Omron Sysmac Studio project OEEF_FS_lib_1_2_2 (Sysmac Studio 1.44.0.64015, LibraryProject)

# Controller new_Controller_0: NX1P2-1040DT1 version 1.21
Task PrimaryTask (priority 4, period or condition 2000): Programme0

TYPE nsAxisControl\eMoveMode : (Relative := 0, Absolute := 1); END_TYPE
TYPE nsAxisControl\eCurveType : (Poly5 := 0, Poly3 := 1, Straight := 2, NoCurve := 9999); END_TYPE
TYPE nsAxisControl\eTypeOfCmd : (CancelMC_Sync := -5, CancelCam := -3, CancelTrack := -2, NoCde := 9999, PolyMvt := 1, Track := 2, Cam := 3, WarmStart := 4, MC_Sync := 5); END_TYPE
TYPE nsAxisControl\stAxisControl : STRUCT
    MasterPosition : nsAxisControl\stMasterPosition;
    MasterAxis : _sAXIS_REF;
    Move : nsAxisControl\stMove;
    Track : nsAxisControl\stTrack;
    Cam : nsAxisControl\stCam;
    Kinematic : nsAxisControl\stKinematic;
    Flags : nsAxisControl\stFlags;
    Monitoring : nsAxisControl\stMonitoring;
    MC_MoveJog : nsAxisControl\stMC_MoveJog;
    MC_SetPosition : nsAxisControl\stMC_SetPosition;
    MC_Power : nsAxisControl\stMC_Power;
    MC_Home : nsAxisControl\stMC_Home;
END_STRUCT END_TYPE
TYPE nsAxisControl\stMC_Power : STRUCT
    Enable : BOOL;
    Status : BOOL;
    Busy : BOOL;
    Error : BOOL;
    ErrorID : WORD;
END_STRUCT END_TYPE
TYPE nsAxisControl\stMC_MoveJog : STRUCT
    PositiveEnable : BOOL;
    NegativeEnable : BOOL;
    Velocity : LREAL;
    Acceleration : LREAL;
    Deceleration : LREAL;
    Busy : BOOL;
    CommandAborted : BOOL;
    Error : BOOL;
    ErrorID : WORD;
END_STRUCT END_TYPE
TYPE nsAxisControl\stMC_SetPosition : STRUCT
    Execute : BOOL;
    Position : LREAL;
    ReferenceType : _eMC_REFERENCE_TYPE;
    Relative : BOOL;
    ExecutionMode : _eMC_EXECUTION_MODE;
    Done : BOOL;
    Busy : BOOL;
    CommandAborted : BOOL;
    Error : BOOL;
    ErrorID : WORD;
END_STRUCT END_TYPE
TYPE nsAxisControl\stMC_Home : STRUCT
    Execute : BOOL;
    Done : BOOL;
    Busy : BOOL;
    CommandAborted : BOOL;
    Error : BOOL;
    ErrorID : WORD;
END_STRUCT END_TYPE
TYPE nsAxisControl\stMasterPosition : STRUCT
    NotFrom_sAXIS_REF : BOOL;
    ExternalVariable : LREAL;
END_STRUCT END_TYPE
TYPE nsAxisControl\stMove : STRUCT
    Pos : LREAL;
    Dist : LREAL;
    Tim : LREAL;
    Accel : LREAL;
    Decel : LREAL;
    PolyType : nsAxisControl\eCurveType;
    Mode : nsAxisControl\eMoveMode;
    SetT_In : LREAL;
    SetT_Out : LREAL;
    T_InDone : BOOL;
    T_OutDone : BOOL;
    Exe : BOOL;
END_STRUCT END_TYPE
TYPE nsAxisControl\stTrack : STRUCT
    Conveyor_Vel : LREAL;
    Pos : LREAL;
    Tim : LREAL;
    TimStop : LREAL;
    Accel : LREAL;
    Decel : LREAL;
    PolyType : nsAxisControl\eCurveType;
    SetT_In : LREAL;
    T_InDone : BOOL;
    Exe : BOOL;
    Cancel : BOOL;
END_STRUCT END_TYPE
TYPE nsAxisControl\stCam : STRUCT
    Profile : ARRAY[0..10] OF nsAxisControl\stNodes;
    FirstProfile : INT;
    WarmStartMasterPos : LREAL;
    WarmStartSlavePos : LREAL;
    WarmStartSlavePosRequest : BOOL;
    Exe : BOOL;
    Cancel : BOOL;
END_STRUCT END_TYPE
TYPE nsAxisControl\stNodes : STRUCT
    Node : ARRAY[0..10] OF nsAxisControl\stNode;
END_STRUCT END_TYPE
TYPE nsAxisControl\stNode : STRUCT
    MasterAxisPos : LREAL;
    SlaveAxisPos : LREAL;
    CurveTypeBefore : nsAxisControl\eCurveType;
    StartingSlope : LREAL;
    EndingSlope : LREAL;
    PreviousProfile : INT;
    NextProfile : INT;
END_STRUCT END_TYPE
TYPE nsAxisControl\stKinematic : STRUCT
    Start : BOOL;
    Stop : BOOL;
    InvKin_in : LREAL;
    InvKin_out : LREAL;
    DirKin_in : LREAL;
    DirKin_out : LREAL;
END_STRUCT END_TYPE
TYPE nsAxisControl\stFlags : STRUCT
    Done : BOOL;
    Synchronising : BOOL;
    Synchronised : BOOL;
END_STRUCT END_TYPE
TYPE nsAxisControl\stMonitoring : STRUCT
    PositioningCmd : LREAL;
    Axis_Act_Pos_MCS : LREAL;
    TypeOfCmd : nsAxisControl\eTypeOfCmd;
    TypeOfCtrlMode : nsAxisControl\eTypeOfCtrlMode;
END_STRUCT END_TYPE
TYPE nsAxisControl\eTypeOfCtrlMode : (ExtKinOff := 0, ExtKinOn := 1, NoCtrlMode := 9999); END_TYPE

TYPE nsKinematics\sKinInOut : STRUCT
    KinSpec : nsKinematics\stSpec;
    Cartesian : nsKinematics\sCartesian;
    Axis : nsKinematics\sAxis;
    KinSize : nsKinematics\stSize;
END_STRUCT END_TYPE
TYPE nsKinematics\stSpec : STRUCT
    KinType : nsKinematics\eKinType;
    KinDir : nsKinematics\eDirInv;
    SCARA : nsKinematics\stSCARA;
END_STRUCT END_TYPE
TYPE nsKinematics\sCartesian : STRUCT
    Cmd_Component : ARRAY[0..2] OF LREAL;
    Act_Component : ARRAY[0..2] OF LREAL;
END_STRUCT END_TYPE
TYPE nsKinematics\sAxis : STRUCT
    A_Cmd : ARRAY[0..9] OF LREAL;
    A_Act : ARRAY[0..9] OF LREAL;
END_STRUCT END_TYPE
TYPE nsKinematics\eKinType : (H_Bot_XY := 0, SCARA := 1); END_TYPE
TYPE nsKinematics\eDirInv : (Direct := 0, Inverse := 1); END_TYPE
TYPE nsKinematics\stSize : STRUCT
    NbOfCoordinates : INT;
    NbOfAxis : INT;
END_STRUCT END_TYPE
TYPE nsKinematics\stSCARA : STRUCT
    Len1 : LREAL;
    Len2 : LREAL;
END_STRUCT END_TYPE

PROGRAM Programme0

(* Section Section0: ladder, written here as Structured Text *)
END_PROGRAM

FUNCTION fPolyTimesNeeded : BOOL
(* Time needed to achieve a movement depending of the curve type and the acceleration or the speed fixed. To do for instance a speed or an acceleration limit. *)
VAR_INPUT
    CurveType : nsAxisControl\eCurveType;
    Distance : LREAL;
    AccDefined : LREAL;
    SpeedDefined : LREAL;
END_VAR
VAR_OUTPUT
    TNeededToAcc : LREAL;
    TNeededToSpeed : LREAL;
END_VAR
(*
*******************************************
*		  Calcule le temps nécessaire			*
*	 pour effectuer un trajet avec une		*
*	accélération ou une vitesse définie		*
*******************************************
*)

CASE CurveType OF
	
	Poly5 :
	// AccDefined exprimée en unité/sec2
	TNeededToAcc:=SQRT(5.8*Distance/AccDefined);

	// SpeedDefined exprimée en unité/sec
	TNeededToSpeed:=1.9*Distance/SpeedDefined;
	
	Poly3 :
	// AccDefined exprimée en unité/sec2
	TNeededToAcc:=SQRT(6*Distance/AccDefined);

	// SpeedDefined exprimée en unité/sec
	TNeededToSpeed:=1.5*Distance/SpeedDefined;
	
END_CASE;
END_FUNCTION

FUNCTION fKinematics : BOOL
(* Normal and inverse tranforms : / - H-Bot XY / - SCARA *)
VAR
    AC : LREAL;
    BAC : LREAL;
    ABC : LREAL;
    angle : LREAL;
    len1 : LREAL;
    len2 : LREAL;
    j2 : LREAL;
    j1 : LREAL;
    x : LREAL;
    y : LREAL;
    z : LREAL;
END_VAR
VAR_IN_OUT
    KinInOut : nsKinematics\sKinInOut;
END_VAR
(*
*******************************************
*		  			Transformées						*
*	 			directes et inverses					*
*******************************************
*)

CASE KinInOut.KinSpec.KinType OF
	(* H-Bot XY *)
	H_Bot_XY :
	KinInOut.KinSize.NbOfCoordinates:=2;				// XY
	KinInOut.KinSize.NbOfAxis:=2;							// A0 et A1

	IF KinInOut.KinSpec.KinDir=Direct THEN
		// Direct
		KinInOut.Cartesian.Act_Component[0]:=(KinInOut.Axis.A_Act[0]+KinInOut.Axis.A_Act[1])*0.5;							// positions actuelle X
		KinInOut.Cartesian.Act_Component[1]:=(KinInOut.Axis.A_Act[0]-KinInOut.Axis.A_Act[1])*0.5;							// positions actuelle Y
	ELSE
		// Inverse
		KinInOut.Axis.A_Cmd[0]:=KinInOut.Cartesian.Cmd_Component[0]+KinInOut.Cartesian.Cmd_Component[1];	// Position de commande axe A0
		KinInOut.Axis.A_Cmd[1]:=KinInOut.Cartesian.Cmd_Component[0]-KinInOut.Cartesian.Cmd_Component[1];	// Position de commande axe A1
	END_IF;	

	(* SCARA *)
	SCARA :
	KinInOut.KinSize.NbOfCoordinates:=3;				// XYZ
	KinInOut.KinSize.NbOfAxis:=3;							// A0 à A2
	
	len1:=KinInOut.KinSpec.SCARA.Len1;					// Longueur du bras
	len2:=KinInOut.KinSpec.SCARA.Len2;					// Longueur de l'avant bras	
	
	IF KinInOut.KinSpec.KinDir=Direct THEN
		// Direct
		j1:=KinInOut.Axis.A_Act[0];								// Angle actuel de l'épaule
		j2:=KinInOut.Axis.A_Act[1];								// Angle actuel du coude
		
		AC:=SQRT(len1*len1+len2*len2-2*len1*len2*COS(DegToRad(j2)));
		BAC:=RadToDeg(ACOS((len1*len1+AC*AC-len2*len2)/(2*len1*AC)));	
		angle:=j1-BAC;
		
		fBaseCoords(AC, angle, KinInOut.Cartesian.Act_Component[0], KinInOut.Cartesian.Act_Component[1]);			// positions actuelles X et Y 
		KinInOut.Cartesian.Act_Component[2]:=KinInOut.Axis.A_Act[2];																		// position actuelle Z 
		
	ELSE
		// Inverse
		x:=KinInOut.Cartesian.Cmd_Component[0];	// Position de commande X
		y:=KinInOut.Cartesian.Cmd_Component[1];	// Position de commande Y
		z:=KinInOut.Cartesian.Cmd_Component[2];	// Position de commande Z
		
		AC:=SQRT(x*x+y*y);
		ABC:=RadToDeg(ACOS((len1*len1+len2*len2-AC*AC)/(2*len1*len2)));
		
		KinInOut.Axis.A_Cmd[0]:=ABC;						// Angle de commande axe 0 (épaule)
		
		IF x>0 AND y>0 THEN										// Angle de commande axe 1 (coude)
			KinInOut.Axis.A_Cmd[1]:=RadToDeg(ACOS(AC/x));
		ELSIF x>0 AND y<0 THEN
			KinInOut.Axis.A_Cmd[1]:=180-RadToDeg(ACOS(AC/x));
		ELSIF x<0 AND y<0 THEN
			KinInOut.Axis.A_Cmd[1]:=180+RadToDeg(ACOS(AC/x));
		ELSE
			KinInOut.Axis.A_Cmd[1]:=360-RadToDeg(ACOS(AC/x));
		END_IF;
		
		KinInOut.Axis.A_Cmd[2]:=z;								// Position de commande axe 2 (vertical)
	END_IF;
END_CASE;
	
END_FUNCTION

FUNCTION fTicksQCalc : LINT
(* Calculation of the quantity of ticks depending of the time of the movement *)
VAR
    TaskPeriod_msec : LINT;
END_VAR
VAR_INPUT
    Tmvt : LREAL;
END_VAR
(*
*******************************************
*		  			Calcul le nombre					*
*	 				de tops d'horloge				*
*******************************************
*)

// Suivant le temps de cycle de la tâche principale
TaskPeriod_msec:= TimeToNanoSec(GetMyTaskInterval())/1000000;

// Suivant le temps du mouvement en secondes
fTicksQCalc:=LREAL_TO_LINT(Tmvt)*1000/TaskPeriod_msec;
END_FUNCTION

FUNCTION fPoly5 : LREAL
(* Polynomial of the 5th order *)
VAR
    a : LREAL;
    b : LREAL;
    c : LREAL;
    d : LREAL;
    e : LREAL;
    f : LREAL;
    K : LREAL;
    xSq : LREAL;
END_VAR
VAR_INPUT
    v0 : LREAL;  (* Vitesse initiale *)
    v1 : LREAL;  (* Vitesse finale *)
    a0 : LREAL;
    a1 : LREAL;
    x : LREAL;
    Offset : LREAL;
    TargetDist : LREAL;
END_VAR
(*
*******************************************
*		  				Polynôme 5						*
*******************************************
*)

// Coéficients 
a:=6.0-3.0*(v0+v1)+((a1-a0)/2.0);
b:=-15.0+8.0*v0+7.0*v1+(3.0*a0/2.0)-a1;
c:=10.0-6.0*v0-4.0*v1-(3.0*a0/2.0)+(a1/2.0);
d:=a0/2.0;
e:=v0;
f:=Offset;
K:=TargetDist;

// Carré de x
xSq:=x*x;

// Position=ax5+bx4+cx3+dx2+ex+f
fPoly5:=f+(K*(a*(xSq*xSq*x)+b*(xSq*xSq)+c*(xSq*x)+d*(xSq)+e*x));
END_FUNCTION

FUNCTION fPoly3 : LREAL
(* Polynomial of the 3th order *)
VAR
    a : LREAL;
    b : LREAL;
    c : LREAL;
    d : LREAL;
    K : LREAL;
    xSq : LREAL;
END_VAR
VAR_INPUT
    v0 : LREAL;  (* Vitesse initiale *)
    v1 : LREAL;  (* Vitesse finale *)
    x : LREAL;
    Offset : LREAL;
    TargetDist : LREAL;
END_VAR
(*
*******************************************
*		  				Polynôme 3						*
*******************************************
*)

// Coéficients 
a:=-2.0+v0+v1;
b:=3.0-2.0*v0-v1;
c:=v0;
d:=Offset;
K:=TargetDist;
		
// Carré de x
xSq:=x*x;

// Position=ax3+bx2+cx+d
fPoly3:=d+(K*(a*(xSq*x)+b*(xSq)+c*x));
END_FUNCTION

FUNCTION fPoly2 : LREAL
(* Polynomial of the 2th order *)
VAR
    a : LREAL;
    b : LREAL;
    c : LREAL;
    xSq : LREAL;
END_VAR
VAR_INPUT
    v0 : LREAL;  (* Vitesse initiale *)
    v1 : LREAL;  (* Vitesse finale *)
    x : LREAL;
    Offset : LREAL;
    TargetDist : LREAL;
END_VAR
(*
*******************************************
*		  				Polynôme 2						*
*******************************************
*)

// Coéfficients
a:=v1-v0;
b:=v0;
c:=Offset;

// Carré de x
xSq:=x*x;

// Position=0,5*ax2+bx+c (primitive d'une droite ax+b)
fPoly2:=(TargetDist*((0.5*a*(xSq)+b*x)))+c;
END_FUNCTION

FUNCTION fStraight : LREAL
(* Straight *)
VAR
    a : LREAL;
    b : LREAL;
END_VAR
VAR_INPUT
    x : LREAL;
    Offset : LREAL;
    TargetDist : LREAL;
END_VAR
(*
*******************************************
*		  					Droite							*
*******************************************
*)

// Coéficients 
a:=TargetDist;
b:=Offset;

// Position=ax+b
fStraight:=a*x+b;
END_FUNCTION

FUNCTION fBaseCoords : BOOL
(* Return coordinates of second joint *)
VAR_INPUT
    length : LREAL;
    angle : LREAL;
END_VAR
VAR_OUTPUT
    x : LREAL;
    y : LREAL;
END_VAR
(*
*******************************************
*		Calcule les coordonnées	XY			*
*		du deuxième joint articulaire			*
*******************************************
*)

IF angle<=90 THEN
	// Premier quadrant
	x:=length*COS(DegToRad(angle));
	y:=length*SIN(DegToRad(angle));
ELSIF angle>90 AND angle<=180 THEN
	// Deuxième quadrant
	x:=-length*COS(DegToRad(180-angle));
	y:=length*SIN(DegToRad(180-angle));
ELSIF angle>180 AND angle<=270 THEN
	// Troisième quadrant
	x:=-length*COS(DegToRad(180-angle));
	y:=-length*SIN(DegToRad(180-angle));
ELSE
	// Quatrième quadrant
	x:=length*COS(DegToRad(360-angle));
	y:=-length*SIN(DegToRad(360-angle));
END_IF;
END_FUNCTION

FUNCTION_BLOCK AxisControl
(* - Cam (multi profiles and Warm start) / - Move abs or rel (pos + time) by polynomials curves (3 & 5) / - Tracking a conveyor / - Blending two axis (T_In & T_Out) / 2. Polynomial 2 for a linear deceleration of the speed in case of track cancelling / 3. Some PLCopen functions nested / 4. Exernal kinematics binding *)
VAR
    FBi_SyncMov : MC_SyncMoveAbsolute;
    FBi_SyncStop : MC_Stop;
    FBe_SetPosition : MC_SetPosition;
    FBe_Home : MC_Home;
    FBi_ReadAxisMasterParam : MC_ReadAxisParameter;
    FBi_ReadAxisSlaveParam : MC_ReadAxisParameter;
    FBe_Power : MC_Power;
    Edge1 : R_TRIG;
    Edge2 : R_TRIG;
    Edge3 : R_TRIG;
    Edge4 : R_TRIG;
    Edge5 : R_TRIG;
    Edge6 : R_TRIG;
    Edge7 : R_TRIG;
    Edge8 : R_TRIG;
    Edge9 : R_TRIG;
    Edge10 : R_TRIG;
    Edge11 : R_TRIG;
    Edge12 : R_TRIG;
    TypeOfCmd : nsAxisControl\eTypeOfCmd;
    TargetDist : LREAL;
    TargetSpeed : LREAL;
    UpExecMvt : BOOL;
    UpExecTrack : BOOL;
    UpExecCam : BOOL;
    UpCancelTrack : BOOL;
    Phase : INT;
    Tick : LINT;
    TicksQ : LINT;
    Offset : LREAL;
    x : LREAL;
    v0 : LREAL;  (* Vitesse initiale *)
    v1 : LREAL;  (* Vitesse finale *)
    LastSpeed : LREAL;
    DistStop : LREAL;
    SyncErr : BOOL;
    SyncErrID : WORD;
    SyncStopErrID : WORD;
    UpKinOn : BOOL;
    UpKinOff : BOOL;
    UpCancelCam : BOOL;
    MasterDistDone : LREAL;
    a1 : LREAL;
    a0 : LREAL;
    FBe_MovJog : MC_MoveJog;
    LastPosSlave : LREAL;
    LastPosMaster : LREAL;
    ReadAxisMasterPParam : _sAXIS_PARAM;
    ReadAxisMasterParameterErr : BOOL;
    ReadAxisMasterParameterErrID : WORD;
    ReadAxisSlavePParam : _sAXIS_PARAM;
    ReadAxisSlaveParameterErr : BOOL;
    ReadAxisSlaveParameterErrID : WORD;
    CamSettingError : BOOL;
    NodesNbMax : INT;
    CurrentSeg : INT;
    Loop : INT;
    X0 : LREAL;
    X1 : LREAL;
    Y0 : LREAL;
    Y1 : LREAL;
    SegmentPolyType : nsAxisControl\eCurveType;
    MasterDist : LREAL;
    SegmentsNb : INT;
    SyncStopErr : BOOL;
    NodesNb : INT;
    UpWarmStartPosReq : BOOL;
    WarmStartCalculation : BOOL;
    v1CamSetting : LREAL;
    v0CamSetting : LREAL;
    Edge10_Q : BOOL;
    Edge10_Clk : BOOL;
    a0CamSetting : LREAL;
    a1CamSetting : LREAL;
    ScannedSeg : INT;
    SetPositionErr : BOOL;
    SetPositionErrID : WORD;
    FBi_SetPosition : MC_SetPosition;
    ProfileToApply : INT := 0;
    ProfilesNb : INT;
    ProfilesNbMax : INT;
    UpCamBeginning : BOOL;
    CamSettingErrorType : STRING[50];
    KinIn : LREAL;
    KinOut : LREAL;
    TypeOfCtrlMode : nsAxisControl\eTypeOfCtrlMode;
    Gen : LREAL;
    Conveyor_Pos : LREAL;
    TaskPeriod_msec_LREAL : LREAL;
    MasterPosition : LREAL;
END_VAR
VAR_INPUT
    Dummy : BOOL;
END_VAR
VAR_OUTPUT
    Error : BOOL;
END_VAR
VAR_IN_OUT CONSTANT
    Axis : _sAXIS_REF;
END_VAR
VAR_IN_OUT
    IO : nsAxisControl\stAxisControl;
END_VAR
VAR_OUTPUT
    ErrorMsg : STRING[80];
END_VAR
(*
*******************************************
*					OEEF - F.SIMON					*
*******************************************
*)

Edge1(IO.Move.Exe,UpExecMvt);															// Commande de mouvement polynômial
Edge2(IO.Track.Exe,UpExecTrack);														// Commande de tracking
Edge3(IO.Track.Cancel,UpCancelTrack);												// Commande d'annulation de tracking
Edge4(IO.Cam.Exe,UpExecCam);															// Commande de mise en came
Edge5(IO.Cam.Cancel,UpCancelCam);													// Commande d'annulation de came
Edge6(IO.Cam.WarmStartSlavePosRequest,UpWarmStartPosReq);		// Commande de Warmstart
Edge7(IO.Kinematic.Start,UpKinOn);													// Commande d'activation de la kinematic
Edge8(IO.Kinematic.Stop,UpKinOff);													// Commande de désactivation de la kinematic


(*
*******************************************
*					Type d'axe maître				*
*******************************************
*)
IF IO.MasterPosition.NotFrom_sAXIS_REF THEN
	MasterPosition:=IO.MasterPosition.ExternalVariable;
ELSE
	MasterPosition:=IO.MasterAxis.Act.Pos;
END_IF;


(*
*******************************************
*		Commande de tracking active		*
*******************************************
*)
IF TypeOfCmd=Track THEN
	// Calcul l'avance du convoyeur
	TaskPeriod_msec_LREAL:= LINT_TO_LREAL(TimeToNanoSec(GetMyTaskInterval())/1000000);
	Conveyor_Pos:=Conveyor_Pos+IO.Track.Conveyor_Vel*(TaskPeriod_msec_LREAL/1000);
	// Polynôme en cours : lecture de la position et de la vitesse du maître pour le raccordement en fin de polynôme
	LastPosMaster:=Conveyor_Pos;					// Position du maître à l'instant
	TargetSpeed:=IO.Track.Conveyor_Vel;			// Vitesse du maître à l'instant
	TargetDist:=LastPosMaster-LastPosSlave; 	// Distance à parcourir depuis l'origine du tracking
	IF IO.Flags.Synchronised THEN
	// Polynôme terminé : synchronisation maître/esclave (following)
		FBi_SyncMov.Position:=Conveyor_Pos;
	END_IF;
END_IF;


(*
*******************************************
*			Commande 	de came					*
*			ou de warmstart active 				*
*******************************************
*)
IF TypeOfCmd=Cam OR TypeOfCmd=WarmStart THEN
	// Profil à appliquer
	Edge9(TRUNC(MasterPosition)=IO.Cam.Profile[ProfileToApply].Node[0].MasterAxisPos,UpCamBeginning);
	IF UpCamBeginning THEN
		IF CurrentSeg=0 THEN
			ProfileToApply:=IO.Cam.Profile[ProfileToApply].Node[0].PreviousProfile; 				// Recule
		ELSE
			ProfileToApply:=IO.Cam.Profile[ProfileToApply].Node[NodesNb-1].NextProfile;	// Avance
		END_IF;
	END_IF;
	
	// Dans le cas d'un WarmStart le profil est imposé car il ne peut être déterminé automatiquement
	IF TypeOfCmd=WarmStart THEN
		ProfileToApply:=IO.Cam.FirstProfile;
	END_IF;

	// Comptage du nombre de noeuds du profil appliqué
	NodesNb:=1;
	WHILE IO.Cam.Profile[ProfileToApply].Node[NodesNb].MasterAxisPos<>0
		DO
		NodesNb:=NodesNb+1;
	END_WHILE;
	
	// Comptage du nombre total de profils
	ProfilesNb:=0;
	REPEAT
		ProfilesNb:=ProfilesNb+1;
	UNTIL IO.Cam.Profile[ProfilesNb].Node[1].MasterAxisPos=0
	END_REPEAT;
	
	// Nombre de segments de la came
	SegmentsNb:=NodesNb-1;
		
	// Evolution du segment en cours
	CASE TypeOfCmd OF
		Cam :
		FOR ScannedSeg:=0 TO SegmentsNb-1 DO
			IF MasterPosition>=IO.Cam.Profile[ProfileToApply].Node[ScannedSeg].MasterAxisPos AND MasterPosition<IO.Cam.Profile[ProfileToApply].Node[ScannedSeg+1].MasterAxisPos THEN
				CurrentSeg:=ScannedSeg;
			END_IF;
		END_FOR;
		WarmStart :
		FOR ScannedSeg:=0 TO SegmentsNb-1 DO
			IF IO.Cam.WarmStartMasterPos>=IO.Cam.Profile[ProfileToApply].Node[ScannedSeg].MasterAxisPos AND IO.Cam.WarmStartMasterPos<IO.Cam.Profile[ProfileToApply].Node[ScannedSeg+1].MasterAxisPos THEN
				CurrentSeg:=ScannedSeg;
			END_IF;
		END_FOR;	
	END_CASE;

	// Paramètres du polynôme dans le segment en cours
	X0:=IO.Cam.Profile[ProfileToApply].Node[CurrentSeg].MasterAxisPos;										// Abscisse de début
	Y0:=IO.Cam.Profile[ProfileToApply].Node[CurrentSeg].SlaveAxisPos;											// Ordonnée de début
	X1:=IO.Cam.Profile[ProfileToApply].Node[CurrentSeg+1].MasterAxisPos;									// Abscisse de fin
	Y1:=IO.Cam.Profile[ProfileToApply].Node[CurrentSeg+1].SlaveAxisPos;									// Ordonnée de fin
	MasterDist:=X1-X0;																														// Distance de la composante X
	TargetDist:=Y1-Y0;																														// Distance de la composante Y
	Offset:=Y0;																																	// Offset de départ

 	CASE TypeOfCmd OF
		Cam : MasterDistDone:=MasterPosition-X0;																			// Distance parcourue par le maître
		WarmStart : MasterDistDone:=IO.Cam.WarmStartMasterPos-X0;
 	END_CASE;
 
	SegmentPolyType:=IO.Cam.Profile[ProfileToApply].Node[CurrentSeg+1].CurveTypeBefore;		// Type de profil
	v0CamSetting:=IO.Cam.Profile[ProfileToApply].Node[CurrentSeg+1].StartingSlope;					// Pente de raccordement de la vitesse de début de segment
	v1CamSetting:=IO.Cam.Profile[ProfileToApply].Node[CurrentSeg+1].EndingSlope;					// Pente de raccordement de la vitesse de fin de segment
	//a0CamSetting:=?																														// Pente de raccordement de l'accélération de début de segment
	//a1CamSetting:=?																														// Pente de raccordement de l'accélération de fin de segment

	// Arrêt du calcul de la position théorique de l'esclave pour le WarmStart
	IF WarmStartCalculation THEN
		WarmStartCalculation:=FALSE;
	END_IF;
END_IF;


(*
*******************************************
*				Mode kinematic actif				*
*******************************************
*)
IF TypeOfCtrlMode=ExtKinOn THEN
	// Envoi le calcul du générateur vers la kinematic
	KinIn:=Gen;
	// Désactive le mode External kinematic en cas d'erreur du MC_SyncMoveAbsolute
	IF FBi_SyncMov.Error THEN
		TypeOfCtrlMode:=NoCtrlMode;
	END_IF;

	// Envoi la commande de position MCS à la kinématic inverse
	IO.Kinematic.InvKin_in:=KinIn;
	// Récupère la commande de position ACS
	KinOut:=IO.Kinematic.InvKin_out;

	// Envoi la position actuelle ACS à la kinématic directe
	IO.Kinematic.DirKin_in:=Axis.Act.Pos;
	// Récupère la position actuelle MCS
	IO.Monitoring.Axis_Act_Pos_MCS:=IO.Kinematic.DirKin_out;
END_IF;


(*
*******************************************
*			Mode kinematic inactif				*
*******************************************
*)
IF TypeOfCtrlMode=ExtKinOff THEN
	// Envoi le calcul du générateur vers la kinematic
	KinIn:=Gen;
	// ACS=MCS
	KinOut:=KinIn;
	IO.Monitoring.Axis_Act_Pos_MCS:=Axis.Act.Pos;
END_IF;


(*
*******************************************
*						Générateur						*
*******************************************
*)
CASE Phase OF
	
	0 : // COMMANDES
	
		// Commande de mouvement polynômial
		IF UpExecMvt AND IO.Move.Tim>0 THEN
			TypeOfCmd:=PolyMvt;
			 // Evite les glitchs
			FBi_SyncMov.Position:=Axis.Act.Pos;
			Gen:=Axis.Act.Pos;
			
			// Nombre de tops d'horloge nécessaires pour le mouvement
			TicksQ:=fTicksQCalc(IO.Move.Tim);
			Tick:=0;
			
			// Calcul de la distance à effectuer
			// Mode kinematic actif
			IF TypeOfCtrlMode=ExtKinOn THEN
				IF IO.Move.Mode=Absolute THEN
					TargetDist:=IO.Move.Pos-IO.Monitoring.Axis_Act_Pos_MCS;
				ELSIF IO.Move.Mode=Relative THEN
					TargetDist:=IO.Move.Dist;
				END_IF;
			ELSE
			// Mode kinematic inactif	
				IF IO.Move.Mode=Absolute THEN
					TargetDist:=IO.Move.Pos-Axis.Act.Pos;
				ELSIF IO.Move.Mode=Relative THEN
					TargetDist:=IO.Move.Dist;
				END_IF;
			END_IF;
			
			Phase:=10;
		END_IF;
		
		// Commande de tracking
		IF UpExecTrack AND IO.Track.Tim>0 AND TypeOfCtrlMode=ExtKinOff THEN
			TypeOfCmd:=Track;
			 // Evite les glitchs
			FBi_SyncMov.Position:=Axis.Act.Pos;
			Gen:=Axis.Act.Pos;
			
			// Le début de tracking fonctionne comme un mouvement polynômial (même polynôme, même temps)
			IO.Move.Tim:=IO.Track.Tim;
			Tick:=0;
			// Nombre de tops d'horloge nécessaires pour le mouvement
			TicksQ:=fTicksQCalc(IO.Move.Tim);
			// Position initiale à tracker
			Conveyor_Pos:=IO.Track.Pos;
			// Dernière position connue de l'esclave
			LastPosSlave:=Axis.Act.Pos;	
			Phase:=10;
		END_IF;
		
		// Annulation du tracking
		IF UpCancelTrack THEN
			TypeOfCmd:=CancelTrack;
			Phase:=30;
		END_IF;

		// Commande de came
		IF UpExecCam THEN
			TypeOfCmd:=Cam;
			 // Evite les glitchs
			FBi_SyncMov.Position:=Axis.Act.Pos;
			Gen:=Axis.Act.Pos;
			
			ProfilesNbMax:=10;
			NodesNbMax:=10;
			ProfileToApply:=IO.Cam.FirstProfile;
			CamSettingError:=FALSE;
			CurrentSeg:=0;
			Phase:=5;
		END_IF;

		// Annulation de la commande de came : Traitée en Phase 20 pendant son exécution

		// Commande de WarmStart
		IF UpWarmStartPosReq THEN
			TypeOfCmd:=WarmStart;
			ProfilesNbMax:=10;
			NodesNbMax:=10;
			ProfileToApply:=IO.Cam.FirstProfile;
			CamSettingError:=FALSE;
			CurrentSeg:=0;
			WarmStartCalculation:=TRUE;
			Phase:=5;
		END_IF;

		// Activation du mode kinematic 
		IF UpKinOn THEN
			TypeOfCtrlMode:=ExtKinOn;
			 // Evite les glitchs
			FBi_SyncMov.Position:=Axis.Act.Pos;
			Gen:=Axis.Act.Pos;
			
			Phase:=100;
		END_IF;
		
		// Désactivation du mode kinematic 
		IF UpKinOff THEN
			TypeOfCtrlMode:=ExtKinOff;
			Phase:=50;
		END_IF;


	5 : // INIT : lecture des paramètres des axes

		FBi_ReadAxisMasterParam.Execute:=TRUE;
		FBi_ReadAxisSlaveParam.Execute:=TRUE;
		
		IF FBi_ReadAxisMasterParam.Done AND FBi_ReadAxisSlaveParam.Done THEN
			FBi_ReadAxisMasterParam.Execute:=FALSE;
			FBi_ReadAxisSlaveParam.Execute:=FALSE;
			Phase:=10;
		END_IF;


	10 : // INIT : flags, offset
	
		// Exe
		FBi_SyncMov.Execute:=FALSE;
	
		// Distance nulle : on ne bouge pas
		IF abs(TargetDist)=0 THEN
			Phase:=0;
		END_IF;
		
		// Flags
		IO.Flags.Synchronising:=FALSE;
		IO.Flags.Synchronised:=FALSE;
		
		// Offsets de départ	
		IF TypeOfCmd<>Cam AND TypeOfCmd<>WarmStart THEN
			// Débute le mouvement à partir de la position actuelle
			// Mode kinematic actif
			IF TypeOfCtrlMode=ExtKinOn THEN
				Offset:=IO.Monitoring.Axis_Act_Pos_MCS;
			ELSE
				Offset:=Axis.Act.Pos;
			END_IF;
			Phase:=15;
		ELSIF TypeOfCmd=Cam THEN
			// Débute le mouvement à partir de Y0
			Offset:=Y0;
			Phase:=15;
		ELSIF TypeOfCmd=WarmStart THEN
			// Débute le mouvement à partir de Y0 et n'active pas la fonction de positionnement cyclique
			Offset:=Y0;
			Phase:=20;
		END_IF;
		
		
	15 : // INIT : activation de la fonction de positionnement cyclique
	
		IF TypeOfCtrlMode=ExtKinOn THEN
			Phase:=20;
		ELSE
(*			 // Evite les glitchs..
			FBi_SyncMov.Position:=Axis.Act.Pos;
			Gen:=Axis.Act.Pos;	*)	
			FBi_SyncMov.Execute:=TRUE;
			
			IF FBi_SyncMov.Active THEN
				FBi_SyncMov.Execute:=FALSE;
				Phase:=20;
			END_IF;
		END_IF;


	20 : // EXECUTION DU PROFIL

		// Flags
		IF TypeOfCmd=Cam THEN
			IO.Flags.Synchronised:=TRUE;		// En came
		ELSE
			IO.Flags.Synchronising:=TRUE;	// hors came
		END_IF;

		// Evolution de x
		IF TypeOfCmd=PolyMvt OR TypeOfCmd=Track THEN
			// En fonction du temps dans l'intervalle [0 ; 1] (hors came)
			x:=LIMIT(0.0,(1.0/LINT_TO_LREAL(TicksQ)*LINT_TO_LREAL(Tick)),1.0);
		ELSIF TypeOfCmd=Cam OR TypeOfCmd=WarmStart THEN
			// En fonction de la distance parcourue par le maître dans l'intervalle [0 ; 1] (En came)
			x:=LIMIT(0.0,((1.0/MasterDist)*MasterDistDone),1.0);
		END_IF;
		
		// Limites du domaine fixées à 0,1 % et 99,9 % du parcours
		IF x<0.001 THEN
			x:=0;
		ELSIF x>0.999 THEN
			x:=1;
		END_IF;
		
		// Vitesses initiale et finale des polynômes 3 et 5
		IF TypeOfCmd=PolyMvt THEN
			 // Fixées à zéro pour un mouvement polynômial
			v0:=0.0;
			v1:=0.0;
		ELSIF TypeOfCmd=Track THEN
			// v1 en continuité avec celle du maître lors d'un tracking : elle est convertie dans l'intervalle [0;1] du polynôme EN COURS
			v0:=0.0;
			v1:=(1/(TargetDist/IO.Move.Tim))*TargetSpeed;
		ELSIF TypeOfCmd=Cam OR TypeOfCmd=WarmStart THEN
			// Imposées par paramétrage de la came
			v0:=v0CamSetting;
			v1:=v1CamSetting;
		END_IF;
		
		// Accélérations initiale et finale du polynôme 5
		IF TypeOfCmd=PolyMvt THEN
			a0:=IO.Move.Accel;
			a1:=IO.Move.Decel;
		ELSIF TypeOfCmd=Track THEN
			a0:=IO.Track.Accel;
			a1:=IO.Track.Decel;
		ELSIF TypeOfCmd=Cam OR TypeOfCmd=WarmStart THEN
			a0:=a0CamSetting;
			a1:=a1CamSetting;
		END_IF;

		// Polynôme 5
		IF (TypeOfCmd=PolyMvt AND IO.Move.PolyType=Poly5
			OR TypeOfCmd=Track AND IO.Track.PolyType=Poly5 
			OR (TypeOfCmd=Cam OR TypeOfCmd=WarmStart) 
			AND SegmentPolyType=Poly5) THEN
			Gen:=fPoly5(v0, v1, a0, a1, x, Offset, TargetDist);

		// Polynôme 3
		ELSIF (TypeOfCmd=PolyMvt AND IO.Move.PolyType=Poly3 
			OR TypeOfCmd=Track AND IO.Track.PolyType=Poly3 
			OR (TypeOfCmd=Cam OR TypeOfCmd=WarmStart) 
			AND SegmentPolyType=Poly3) THEN
			Gen:=fPoly3(v0, v1, x, Offset, TargetDist);

		// Straight
		ELSIF  (TypeOfCmd=PolyMvt AND IO.Move.PolyType=Straight 
			OR TypeOfCmd=Track AND IO.Track.PolyType=Straight 
			OR (TypeOfCmd=Cam OR TypeOfCmd=WarmStart) 
			AND SegmentPolyType=Straight) THEN
			Gen:=fStraight(x, Offset, TargetDist);
		END_IF;

		// Suivi de l'évolution du temps (hors came)
		IF TypeOfCmd=PolyMvt OR TypeOfCmd=Track THEN
			IF Tick<TicksQ THEN
				Tick:=Tick+1;
	 		// Fin du polynome dans le cas d'une commande de type tracking
			ELSIF TypeOfCmd=Track THEN
				IO.Flags.Synchronised:=TRUE;
				IO.Flags.Synchronising:=FALSE;
				Phase:=0;
		 	// Fin du polynome dans le cas d'une commande de mouvement polynômial
			ELSIF TypeOfCmd=PolyMvt THEN
				IF TypeOfCtrlMode=ExtKinOff THEN
					IO.Flags.Synchronising:=FALSE; 
					Phase:=50;
				ELSE
					// En mode External kinematic on reste synchronisé
					Phase:=0;
				END_IF;
			END_IF;
		// Suivi de l'évolution du maître (en came)
		ELSIF TypeOfCmd=Cam THEN			
			// Arrêt
			IF UpCancelCam THEN
				IO.Flags.Synchronised:=FALSE;
				Phase:=50;
			END_IF;
		// Calcul de la position théorique de l'esclave pour le WarmStart
		ELSIF TypeOfCmd=WarmStart THEN
			// Le calcul est terminé
			IO.Cam.WarmStartSlavePos:=Gen;
			IF NOT WarmStartCalculation THEN
				Phase:=0;
			END_IF;
		END_IF;
		
	
	30 : // INIT DECELERATION LINEAIRE
		
		Tick:=0;
		TicksQ:=fTicksQCalc(IO.Track.TimStop);	// Nombre de tops d'horloge nécessaires pour le mouvement
		LastSpeed:=TargetSpeed; 						// Dernière vitesse connue avant le prochain polynôme
		IO.Flags.Synchronised:=FALSE;
		Phase:=40;
		
		
	40 : // DECELERATION LINEAIRE
		
		// Evolution de x en fonction du temps dans l'intervalle [0 ; 1]
		x:=LINT_TO_LREAL(Tick)*(1.0/LINT_TO_LREAL(TicksQ));

		// Calcul de la distance d'arrêt en fonction du temps imparti : la distance est divisée par deux car la vitesse diminue de manière linéaire jusqu'à zéro
		DistStop:=(LastSpeed*IO.Track.TimStop)/2;
		
		// Vitesse initiale en continuité avec la dernière vitesse connue : cette vitesse est convertie dans l'intervalle [0;1] du nouveau polynôme
		v0:=(1/(DistStop/IO.Track.TimStop))*LastSpeed;
		
		// Vitesse finale fixée à zéro
		v1:=0.0;
		
		TargetDist:=DistStop;		// Distance d'arrêt
		
		Offset:=LastPosMaster;	// Position initiale en continuité avec la dernière position connue du maître
		
		FBi_SyncMov.Position:=fPoly2(v0, v1, x, Offset, TargetDist);
		
		// Evolution du temps
		IF Tick<TicksQ THEN
			Tick:=Tick+1;
		ELSE
			// Fin du polynôme
			Phase:=50;
		END_IF;
		
		
	50 : // DECONNEXION
	
		FBi_SyncStop.Execute:=TRUE;

		IF FBi_SyncStop.Done THEN
			FBi_SyncStop.Execute:=FALSE;
			Phase:=0;
		END_IF;
		
		
	100 : // CONNEXION
	
		FBi_SyncMov.Position:=Axis.Act.Pos; // Evite les glitchs..
		FBi_SyncMov.Execute:=TRUE;
		
		IF FBi_SyncMov.Active THEN
			FBi_SyncMov.Execute:=FALSE;
			Phase:=0;
		END_IF;
	
END_CASE;


(*
*******************************************
*						Drapeaux							*
*******************************************
*)
// Délai atteint après le début d'un mouvement polynômial ou d'un tracking
IF TypeOfCmd=PolyMvt THEN
	Edge10_Clk:=Tick>=fTicksQCalc(IO.Move.SetT_In);
ELSIF TypeOfCmd=Track THEN
	Edge10_Clk:=Tick>=fTicksQCalc(IO.Track.SetT_In);
END_IF;
Edge10(Edge10_Clk,Edge10_Q);
IF TypeOfCmd=PolyMvt THEN
	IO.Move.T_InDone:=Edge10_Q;
ELSIF TypeOfCmd=Track THEN
	IO.Track.T_InDone:=Edge10_Q;
END_IF;

// Délai atteint avant la fin d'un mouvement polynômial
Edge11((Tick>=(TicksQ-fTicksQCalc(IO.Move.SetT_Out))),IO.Move.T_OutDone);

// Done
Edge12(Phase=0,IO.Flags.Done);
IF IO.Flags.Done THEN
	TypeOfCmd:=NoCde;
END_IF;


(*
*******************************************
*							Erreurs							*
*******************************************
*)
	// Erreur : le nombre de noeuds est supérieur au maximum autorisé
	IF NodesNb>NodesNbMax THEN
		CamSettingError:=TRUE;
		CamSettingErrorType:='Too much nodes'; 
		Phase:=0;
	END_IF;
	
	// Erreur : le nombre de profils est supérieur au maximum autorisé
	IF ProfilesNb>ProfilesNbMax THEN
		CamSettingError:=TRUE;
		CamSettingErrorType:='Too much profiles';
		Phase:=0;
	END_IF;
	
	// Erreur : une valeur maximale de modulo de l'axe maître a été franchie
	IF IO.MasterAxis.Scale.CountMode=_mcCountModeRotary THEN
		FOR Loop:=0 TO NodesNb DO
			IF IO.Cam.Profile[ProfileToApply].Node[Loop].MasterAxisPos>IO.MasterAxis.Scale.MaxPos OR
				IO.Cam.Profile[ProfileToApply].Node[Loop].MasterAxisPos<IO.MasterAxis.Scale.MinPos THEN
				CamSettingError:=TRUE;
				CamSettingErrorType:='Master MaxPos or MinPos overflow';
				Phase:=0;
			END_IF;
		END_FOR;
	END_IF;
	
	// Erreur : une valeur maximale de modulo de l'axe esclave a été franchie
	IF Axis.Scale.CountMode=_mcCountModeRotary THEN
		FOR Loop:=0 TO NodesNb DO
			IF 	IO.Cam.Profile[ProfileToApply].Node[Loop].SlaveAxisPos>Axis.Scale.MaxPos OR
				IO.Cam.Profile[ProfileToApply].Node[Loop].SlaveAxisPos<Axis.Scale.MinPos THEN
				CamSettingError:=TRUE;
				CamSettingErrorType:='Slave MaxPos or MinPos overflow';
				Phase:=0;
			END_IF;
		END_FOR;
	END_IF;
	
	// Erreur : une limite logicielle de l'axe maître a été franchie
	IF ReadAxisMasterPParam.Limit.SwLimitMode<>_mcNonSwLmt THEN
		FOR Loop:=0 TO NodesNb DO
			IF 	IO.Cam.Profile[ProfileToApply].Node[Loop].MasterAxisPos>ReadAxisMasterPParam.Limit.PosiSwLimit OR
				IO.Cam.Profile[ProfileToApply].Node[Loop].MasterAxisPos<ReadAxisMasterPParam.Limit.NegaSwLimit THEN
				CamSettingError:=TRUE;
				CamSettingErrorType:='Master software limit overflow';
				Phase:=0;
			END_IF;
		END_FOR;
	END_IF;
	
	// Erreur : une limite logicielle de l'axe esclave a été franchie
	IF ReadAxisSlavePParam.Limit.SwLimitMode<>_mcNonSwLmt THEN
		FOR Loop:=0 TO NodesNb DO
			IF 	IO.Cam.Profile[ProfileToApply].Node[Loop].SlaveAxisPos>ReadAxisSlavePParam.Limit.PosiSwLimit OR
				IO.Cam.Profile[ProfileToApply].Node[Loop].SlaveAxisPos<ReadAxisSlavePParam.Limit.NegaSwLimit THEN
				CamSettingError:=TRUE;
				CamSettingErrorType:='Slave software limit overflow';
				Phase:=0;
			END_IF;
		END_FOR;
	END_IF;

// Drapeau d'erreur
IF SyncErr OR SyncStopErr OR ReadAxisMasterParameterErr OR ReadAxisSlaveParameterErr OR CamSettingError OR	// Erreurs internes
	IO.MC_Power.Error OR IO.MC_MoveJog.Error OR IO.MC_SetPosition.Error THEN															// Erreurs externes
	Error:=TRUE;
	Phase:=0;
ELSE
	Error:=FALSE;
END_IF;

// Message d'erreur
IF SyncErr THEN
	ErrorMsg:='Internal error : MC_SyncMoveAbsolute';
ELSIF
	SyncStopErr THEN
	ErrorMsg:='Internal error : MC_Stop';
ELSIF
	ReadAxisMasterParameterErr THEN
	ErrorMsg:='Internal error : MC_ReadAxisParameter master';
ELSIF
	ReadAxisSlaveParameterErr THEN
	ErrorMsg:='Internal error : MC_ReadAxisParameter slave';
ELSIF
	CamSettingError THEN
	ErrorMsg:=CONCAT('Internal error : Cam setting error ',CamSettingErrorType);
ELSIF
	IO.MC_Power.Error THEN
	ErrorMsg:='External error : MC_Power';
ELSIF
	IO.MC_MoveJog.Error THEN
	ErrorMsg:='External error : MC_MoveJog';
ELSIF
	IO.MC_SetPosition.Error THEN
	ErrorMsg:='External error : MC_SetPosition';
ELSE
	ClearString(ErrorMsg);
END_IF;
	

(*
*******************************************
*						Monitoring						*
*******************************************
*)
IO.Monitoring.PositioningCmd:=FBi_SyncMov.Position;
IO.Monitoring.TypeOfCmd:=TypeOfCmd;
IO.Monitoring.TypeOfCtrlMode:=TypeOfCtrlMode;


(*
*******************************************
*				Fonctions internes					*
*******************************************
*)
// Positionnement cyclique

// Gestion du modulo
IF Axis.Scale.CountMode=_mcCountModeRotary THEN
	IF KinOut>=Axis.Scale.MaxPos THEN
		FBi_SyncMov.Position:=Axis.Scale.MaxPos-1e-6;		// On s'approche de MaxPos sinon défaut MC_SyncMoveAbs
	ELSIF KinOut<=Axis.Scale.MinPos THEN
		FBi_SyncMov.Position:=Axis.Scale.MinPos;				// On ne dépasse pas MinPos sinon défaut Out of range
	ELSE
		FBi_SyncMov.Position:=KinOut;
	END_IF;
	// Passage du modulo
	FBi_SyncMov.Direction:=_mcShortestWay;
ELSE
	// Axe en mode linéaire
	FBi_SyncMov.Direction:=_mcNoDirection;
	FBi_SyncMov.Position:=KinOut;
END_IF;
		
FBi_SyncMov(
					Axis:=							Axis, 
					// Execute:=, 
					// Position:=, 
					// Direction:=,
					BufferMode:=				_mcAborting, 
					// InPosition=>, 
					// Busy=>,
					// Active=>,
					// CommandAborted=>,
					Error=>						SyncErr, 
					ErrorID=>					SyncErrID
					);

// Arrêt du positionnement cyclique
FBi_SyncStop(
					Axis:=							Axis, 
					// Execute:=, 
					// Deceleration:=, 
					// Jerk:=, 
					// BufferMode:=, 
					// Done=>, 
					// Busy=>, 
					// Active=>, 
					// CommandAborted=>, 
					Error=> 						SyncStopErr,
					ErrorID=>					SyncStopErrID
					);

// Lecture des paramètres de l'axe maître
FBi_ReadAxisMasterParam(
					Axis:=IO.MasterAxis,
					AxisParameter:=ReadAxisMasterPParam,
					// Execute:=,
					// Done=>,
					// Busy=>,
					// CommandAborted=>,
					Error=>ReadAxisMasterParameterErr,
					ErrorID=>ReadAxisMasterParameterErrID
					);

// Lecture des paramètres de l'axe esclave
FBi_ReadAxisSlaveParam(
					Axis:=Axis,
					AxisParameter:=ReadAxisSlavePParam,
					// Execute:=,
					// Done=>,
					// Busy=>,
					// CommandAborted=>,
					Error=>ReadAxisSlaveParameterErr,
					ErrorID=>ReadAxisSlaveParameterErrID
					);

// MC_SetPosition
FBi_SetPosition(
					Axis:=Axis,
					// Execute:=, 
					// Position:=, 
					// ReferenceType:=, 
					// Relative:=, 
					// ExecutionMode:=, 
					// Done=>, 
					// Busy=>, 
					// CommandAborted=>, 
					Error=>SetPositionErr, 
					ErrorID=>SetPositionErrID
					);


(*
*******************************************
*				Fonctions externes					*
*******************************************
*)
// MC_Power
FBe_Power(
				Axis:=Axis, 
				Enable:=IO.MC_Power.Enable, 
				Status=>IO.MC_Power.Status, 
				Busy=>IO.MC_Power.Busy, 
				Error=>IO.MC_Power.Error, 
				ErrorID=>IO.MC_Power.ErrorID
				);

// MC_MoveJog
FBe_MovJog(
					Axis:= Axis,
					PositiveEnable:=IO.MC_MoveJog.PositiveEnable, 
					NegativeEnable:=IO.MC_MoveJog.NegativeEnable, 
					Velocity:=IO.MC_MoveJog.Velocity, 
					Acceleration:=IO.MC_MoveJog.Acceleration, 
					Deceleration:=IO.MC_MoveJog.Deceleration,
					Busy=>IO.MC_MoveJog.Busy, 
					CommandAborted=>IO.MC_MoveJog.CommandAborted, 
					Error=>IO.MC_MoveJog.Error, 
					ErrorID=>IO.MC_MoveJog.ErrorID
					);

// MC_SetPosition
FBe_SetPosition(
					Axis:=Axis,
					Execute:=IO.MC_SetPosition.Execute, 
					Position:=IO.MC_SetPosition.Position, 
					ReferenceType:=IO.MC_SetPosition.ReferenceType, 
					Relative:=IO.MC_SetPosition.Relative, 
					ExecutionMode:=IO.MC_SetPosition.ExecutionMode, 
					Done=>IO.MC_SetPosition.Done, 
					Busy=>IO.MC_SetPosition.Busy, 
					CommandAborted=>IO.MC_SetPosition.CommandAborted, 
					Error=>IO.MC_SetPosition.Error, 
					ErrorID=>IO.MC_SetPosition.ErrorID
					);

// MC_Home
FBe_Home(
					Axis:=Axis,
					Execute:=IO.MC_Home.Execute, 
					Done=>IO.MC_Home.Done, 
					Busy=>IO.MC_Home.Busy, 
					CommandAborted=>IO.MC_Home.CommandAborted, 
					Error=>IO.MC_Home.Error, 
					ErrorID=>IO.MC_Home.ErrorID
					);
END_FUNCTION_BLOCK

FUNCTION_BLOCK KinOnOff
(* Choosing and enabling an external kinematic *)
VAR
    Edge1 : R_TRIG;
    Edge2 : F_TRIG;
    UpKinOn : BOOL;
    DownKinOn : BOOL;
    loop : INT;
END_VAR
VAR_INPUT
    KinON : BOOL;
    NbOfAxis : INT;
END_VAR
VAR_IN_OUT
    Axis_Control : ARRAY[0..9] OF nsAxisControl\stAxisControl;
END_VAR
VAR_OUTPUT
    KinON_status : BOOL;
END_VAR
(*
*******************************************
*		 Active/Désactive la kinematic			*
*******************************************
*)

// Fronts
Edge1(KinON,UpKinOn);
Edge2(KinON,DownKinOn);

// Activation de la kinematic
IF UpKinOn THEN
	FOR loop:=0 TO NbOfAxis-1 DO
		Axis_Control[loop].Kinematic.Start:=TRUE;
		Axis_Control[loop].Kinematic.Stop:=FALSE;
	END_FOR;
END_IF;

// Désactivation de la kinematic
IF DownKinOn THEN
	FOR loop:=0 TO NbOfAxis-1 DO
		Axis_Control[loop].Kinematic.Stop:=TRUE;
		Axis_Control[loop].Kinematic.Start:=FALSE;
	END_FOR;
END_IF;

// Etat
KinON_status:=TRUE;
FOR loop:=0 TO NbOfAxis-1 DO
	IF 	Axis_Control[loop].Monitoring.TypeOfCtrlMode=ExtKinOff THEN
		KinON_status:=FALSE;
	END_IF;
END_FOR;
END_FUNCTION_BLOCK

FUNCTION_BLOCK AverageFilter
VAR
    Loop : INT;
    Samples : ARRAY[0..99] OF LREAL;
    Sum : LREAL;
END_VAR
VAR_INPUT
    Dummy : BOOL;
END_VAR
VAR_OUTPUT
    Ok : BOOL;
END_VAR
VAR_INPUT
    Measure : LREAL;
    QofSamples : INT;
END_VAR
VAR_OUTPUT
    Result : LREAL;
END_VAR
(*
*******************************************
*		   Filtre à moyenne glissante			*
*******************************************
*)

Loop:=1;
REPEAT
	// Pousse la pile pour libérer le premier rang
	Samples[QofSamples-Loop]:=Samples[QofSamples-(Loop+1)];
	Loop:=Loop+1;
UNTIL Loop>=QofSamples
END_REPEAT;
// Place le nouvel échantillon au premier rang
Samples[0]:=Measure;
Loop:=1;
Sum:=0.0;
REPEAT
	// Calcul la somme des échantillons
	Sum:=Sum+Samples[Loop-1];
	Loop:=Loop+1;
UNTIL Loop>QofSamples
END_REPEAT;
// Calcul la moyenne
Result:=Sum/QofSamples;
END_FUNCTION_BLOCK